FUNCTION TFCheckLayerPresence : INT
VAR_INPUT
	WorkArea : POINTER TO ARRAY [1..MAXAREA] OF TFMachinePalletizer_WorkArea;
	WorkAreaState : POINTER TO ARRAY [1..MAXAREA] OF TFMachinePalletizer_WorkAreaState;
	PX_WorkArea : ARRAY [1..MAXAREA] OF BOOL;
END_VAR
VAR
	NStack : INT;
	i : UINT;
END_VAR

TFCheckLayerPresence := 0;
NStack := 0;

FOR i:=1 TO MAXAREAPRESENT DO
	IF WorkArea^[i].Enable = 1 AND WorkArea^[i].Typology = TYPOLOGY_LAYER AND (*WorkAreaState^[i].State = WORKAREA_STATE_OCCUPIED_WORKING*)  PX_WorkArea[i] THEN
		RETURN;
	END_IF
END_FOR
TFCheckLayerPresence := 1;

END_FUNCTION

(* stored: Version 1.1.0.1, ProductVersion 3.1.4024.11
   POU TFCheckLayerPresence: Id {b9005176-eeb3-466f-bded-8b1f1544ddbe}, SpecialFunc None *)
